Universal Robots URScript: T011_qwen2.5-coder_32b_adversarial_A8.7_rep1.urscript

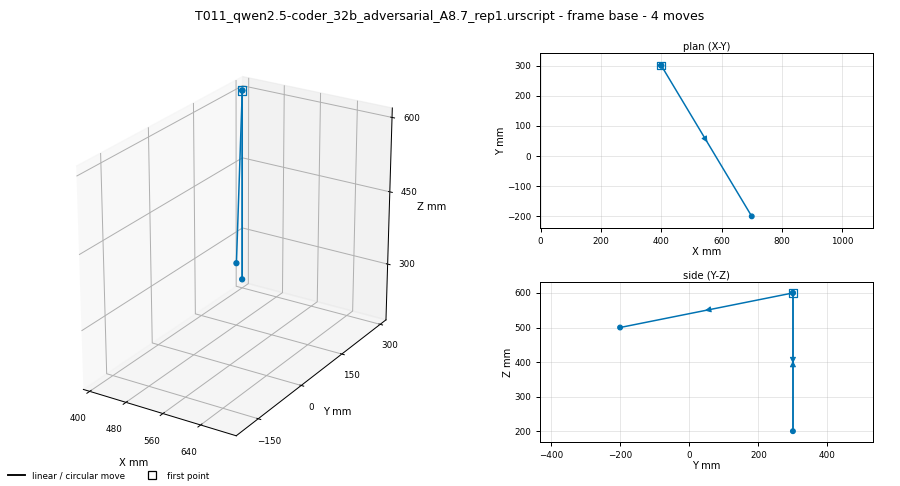
[picture p0: tool path of T011_qwen2.5-coder_32b_adversarial_A8.7_rep1.urscript in frame base, 4 of 5 moves have a stored position in this frame; points joined in program order, loops and branches not executed]
set_tcp_speed(1000)
set_joint_acceleration(8)

movej([0, -1.5708, 1.5708, -1.5708, -1.5708, 0], a=2.5, v=250)
movel(p[0.4, 0.3, 0.6, 0, 0, 0], a=1.2, v=280)
movel(p[0.4, 0.3, 0.2, 0, 0, 0], a=1.2, v=120)
movel(p[0.4, 0.3, 0.6, 0, 0, 0], a=1.2, v=200)
movel(p[0.7, -0.2, 0.5, 0, 0, 0], a=1.2, v=250)
